// TIA Portal V17 export
// export: Created 2023-04-11T11:40:01.3872318Z, ExportSetting WithDefaults, DisplayName Totally Integrated Automation Portal, DisplayVersion V17 Update 3, DisplayName TIA Portal Openness, DisplayVersion V17 Update 3, DisplayName TIA Portal Version Control Interface, DisplayVersion V17, DisplayName SINAMICS Startdrive Advanced, DisplayVersion V17 Update2, DisplayName SINAMICS Startdrive G130, G150, S120, S150, SINAMICS MV, S210, DisplayVersion V17 Update2, DisplayName SINAMICS Startdrive G110M, G120, G120C, G120D, G120P, G115D, DisplayVersion V17 Update2, DisplayName STEP 7 Professional, DisplayVersion V17 Update 3, DisplayName STEP 7 Safety, DisplayVersion V17, DisplayName WinCC UA Professional, DisplayVersion V17 Update 3
TYPE "t_DT_MB_CLIENT_INPUT"
// stored: IsFailsafeCompliant false
   STRUCT
      REQ { ExternalVisible := 'False'} : Bool;   // Activates the requested transmission if TRUE
      DISCONNECT { ExternalVisible := 'False'} : Bool;   // Initiates a disconnect operation
      MB_MODE { ExternalVisible := 'False'} : USInt;   // Specifies the type of request: read, write or diagnostic
      MB_DATA_ADDR { ExternalVisible := 'False'} : UDInt;   // Specifies the starting address of the data to be accessed in the Modbus client
      MB_DATA_LEN { ExternalVisible := 'False'} : UInt;   // Specifies the number of bits or words to be accessed
   END_STRUCT;
END_TYPE
